(* IEC 61131-3 sources: Building-Automation/, 2 files *)

(* ---- global_vars.st ---- *)
(*
===============================================
GLOBAL VARIABLE DECLARATIONS
===============================================
This file contains all global variables, constants,
and type definitions for the PLC project.
*)

VAR_GLOBAL
    // System status variables
    SystemVersion       : STRING := 'PLC_Control_v1.0';
    SystemStartTime     : TIME;
    TotalRunHours       : REAL := 0.0;

    // Production statistics
    TotalCycles         : DINT := 0;
    SuccessfulCycles    : DINT := 0;
    FailedCycles        : DINT := 0;
    ProductionRate      : REAL := 0.0;     // Cycles per hour

    // System configuration
    AutoMode            : BOOL := TRUE;     // Auto/Manual mode
    MaintenanceMode     : BOOL := FALSE;    // Maintenance mode flag

    // Communication status
    HMI_Connected       : BOOL := FALSE;    // HMI connection status
    SCADA_Connected     : BOOL := FALSE;    // SCADA connection status
END_VAR

VAR_GLOBAL CONSTANT
    // Physical constants
    MAX_TEMPERATURE     : REAL := 120.0;    // Maximum safe temperature (°C)
    MIN_TEMPERATURE     : REAL := 10.0;     // Minimum operating temperature (°C)
    MAX_PRESSURE        : REAL := 10.0;     // Maximum system pressure (bar)

    // Timing constants
    STARTUP_DELAY       : TIME := T#5S;     // System startup delay
    SHUTDOWN_DELAY      : TIME := T#3S;     // System shutdown delay
    ALARM_DELAY         : TIME := T#1S;     // Alarm activation delay

    // Control parameters
    DEFAULT_TEMP_SP     : REAL := 75.0;     // Default temperature setpoint
    TEMP_DEADBAND       : REAL := 1.0;      // Temperature control deadband

    // I/O addresses (symbolic names)
    // Digital inputs
    DI_START_BUTTON     : STRING := '%I0.0';
    DI_STOP_BUTTON      : STRING := '%I0.1';
    DI_EMERGENCY_STOP   : STRING := '%I0.2';
    DI_LEVEL_SENSOR     : STRING := '%I0.3';

    // Analog inputs
    AI_TEMPERATURE      : STRING := '%IW0';
    AI_PRESSURE         : STRING := '%IW2';

    // Digital outputs
    DO_PUMP             : STRING := '%Q0.0';
    DO_HEATER           : STRING := '%Q0.1';
    DO_VALVE_1          : STRING := '%Q0.2';
    DO_VALVE_2          : STRING := '%Q0.3';
    DO_ALARM_LIGHT      : STRING := '%Q0.4';
    DO_STATUS_LIGHT     : STRING := '%Q0.5';
END_VAR

(*
===============================================
USER DEFINED TYPES
===============================================
*)

TYPE SystemState : (
    STOPPED := 0,
    STARTING := 1,
    RUNNING := 2,
    STOPPING := 3,
    FAULT := 4,
    MAINTENANCE := 5
);
END_TYPE

TYPE AlarmLevel : (
    NO_ALARM := 0,
    WARNING := 1,
    ALARM := 2,
    CRITICAL := 3
);
END_TYPE

TYPE ProcessData : STRUCT
    Temperature         : REAL;
    Pressure           : REAL;
    FlowRate           : REAL;
    Level              : REAL;
    Timestamp          : DATE_AND_TIME;
END_STRUCT;
END_TYPE

(* ---- main.st ---- *)
PROGRAM Main
VAR
    // Input variables - typically mapped to physical I/O
    StartButton     : BOOL := FALSE;    // I0.0 - Start button
    StopButton      : BOOL := FALSE;    // I0.1 - Stop button
    EmergencyStop   : BOOL := FALSE;    // I0.2 - Emergency stop
    LevelSensor     : BOOL := FALSE;    // I0.3 - Tank level sensor
    TempSensor      : REAL := 20.0;     // IW0 - Temperature sensor (°C)
    PressureSensor  : REAL := 0.0;      // IW2 - Pressure sensor (bar)

    // Output variables - typically mapped to physical outputs
    Pump            : BOOL := FALSE;    // Q0.0 - Main pump
    Heater          : BOOL := FALSE;    // Q0.1 - Heating element
    Valve1          : BOOL := FALSE;    // Q0.2 - Inlet valve
    Valve2          : BOOL := FALSE;    // Q0.3 - Outlet valve
    AlarmLight      : BOOL := FALSE;    // Q0.4 - Red alarm light
    StatusLight     : BOOL := FALSE;    // Q0.5 - Green status light

    // Internal variables
    SystemRunning   : BOOL := FALSE;    // System state flag
    SystemReady     : BOOL := FALSE;    // System ready flag
    AlarmActive     : BOOL := FALSE;    // Alarm state
    CycleCount      : INT := 0;         // Production cycle counter

    // Setpoints and parameters
    SetTemperature  : REAL := 75.0;     // Temperature setpoint (°C)
    MaxPressure     : REAL := 5.0;      // Maximum pressure limit (bar)
    TempTolerance   : REAL := 2.0;      // Temperature tolerance (°C)

    // Timers
    StartupTimer    : TON;              // Startup delay timer
    HeatingTimer    : TON;              // Heating cycle timer
    PumpTimer       : TON;              // Pump run timer
    AlarmTimer      : TON;              // Alarm delay timer

    // Function block instances
    TempController  : PID_Controller;   // Temperature PID controller
END_VAR

// ===============================================
// MAIN PROGRAM LOGIC
// ===============================================

// System safety checks
SystemReady := NOT EmergencyStop AND
               LevelSensor AND
               (PressureSensor < MaxPressure) AND
               NOT AlarmActive;

// Start/Stop logic
IF StartButton AND SystemReady AND NOT SystemRunning THEN
    SystemRunning := TRUE;
    CycleCount := CycleCount + 1;
END_IF;

IF StopButton OR EmergencyStop OR AlarmActive THEN
    SystemRunning := FALSE;
END_IF;

// ===============================================
// PROCESS CONTROL LOGIC
// ===============================================

IF SystemRunning THEN
    // Startup sequence with delay
    StartupTimer(IN := TRUE, PT := T#2S);

    IF StartupTimer.Q THEN
        // Open inlet valve
        Valve1 := TRUE;

        // Start pump after valve opens
        PumpTimer(IN := TRUE, PT := T#1S);
        IF PumpTimer.Q THEN
            Pump := TRUE;
        END_IF;

        // Temperature control
        IF TempSensor < (SetTemperature - TempTolerance) THEN
            Heater := TRUE;
            HeatingTimer(IN := TRUE, PT := T#30S);
        ELSIF TempSensor > (SetTemperature + TempTolerance) THEN
            Heater := FALSE;
            HeatingTimer(IN := FALSE);
        END_IF;

        // Process completion check
        IF TempSensor >= SetTemperature AND HeatingTimer.Q THEN
            Valve2 := TRUE;  // Open outlet valve
        END_IF;

    END_IF;

ELSE
    // System stopped - reset all outputs
    StartupTimer(IN := FALSE);
    PumpTimer(IN := FALSE);
    HeatingTimer(IN := FALSE);
    Pump := FALSE;
    Heater := FALSE;
    Valve1 := FALSE;
    Valve2 := FALSE;
END_IF;

// ===============================================
// ALARM LOGIC
// ===============================================

// Check for alarm conditions
AlarmActive := (PressureSensor > MaxPressure) OR
               (TempSensor > 100.0) OR
               (SystemRunning AND NOT LevelSensor);

// Alarm timer for debouncing
AlarmTimer(IN := AlarmActive, PT := T#500MS);

IF AlarmTimer.Q THEN
    AlarmLight := TRUE;
    SystemRunning := FALSE;  // Emergency shutdown
ELSE
    AlarmLight := FALSE;
END_IF;

// ===============================================
// STATUS INDICATORS
// ===============================================

// Status light shows system ready and running
StatusLight := SystemReady AND SystemRunning;

// Reset alarm when conditions clear
IF NOT AlarmActive AND NOT SystemRunning THEN
    AlarmActive := FALSE;
END_IF;

END_PROGRAM
